Omron CX-Programmer project 新工程 (CX-Programmer 9.73)

# PLC 新PLC1: CS1G-H CPU43

## Global symbols (name address type ; comment)
0.00 BOOL  ; 高压电机启动SB201
0.01 BOOL  ; 高压电机停止SB202
0.02 BOOL  ; 1#高压水泵启动SB203
0.03 BOOL  ; 1#高压水泵停止SB204
0.04 BOOL  ; 1#高压水泵下限SP201
0.05 BOOL  ; 2#高压水泵启动SB205
0.06 BOOL  ; 2#高压水泵停止SB206
0.07 BOOL  ; 2#高压水泵下限SP202
0.08 BOOL  ; 1#润滑油泵启动SB207
0.09 BOOL  ; 1#润滑油泵停止SB208
0.10 BOOL  ; 2#润滑油泵启动SB209
0.11 BOOL  ; 2#润滑油泵停止SB210
0.12 BOOL  ; 前轴承流量下限SP203
0.13 BOOL  ; 后轴承流量下限SP204
0.14 BOOL  ; 前轴承温度上限SP201
0.15 BOOL  ; 后轴承温度上限ST202
100.00 BOOL  ; 断电释放
10.00 BOOL  ; 排料三通阀YV209
10.01 BOOL  ; 防反喷阀进YV203
10.02 BOOL  ; 防反喷阀退YV204
10.03 BOOL  ; 1#断电释放阀YV205
10.04 BOOL  ; 2#断电释放阀YV206
10.05 BOOL  ; 1#蓄压器冲压阀YV207
10.06 BOOL  ; 2#蓄压器冲压阀YV208
10.07 BOOL  ; 搅拌桶下胶电磁阀
10.08 BOOL  ; 1#振动电机M213
10.09 BOOL  ; 原胶搅拌电机M215
10.10 BOOL  ; 输胶泵KA27控制制胶启停
10.12 BOOL  ; 施蜡电机M
10.13 BOOL  ; 施胶泵BPM218
10.14 BOOL  ; 干燥风机停止KA31
10.15 BOOL  ; 干燥风机运行指示
110.00 BOOL  ; Y料位计数启动位
110.05 BOOL  ; 高限料位计数器复
114 CHANNEL  ; 高限料位数据通道
11.00 BOOL  ; 干燥风机电机运行
11.01 BOOL  ; 风机转阀故障灯
11.02 BOOL  ; 干燥风机转阀I
11.03 BOOL  ; 调偏阀2
11.04 BOOL  ; 排污阀
11.05 BOOL  ; 调偏阀1
11.06 BOOL  ; 防火皮带正转
11.07 BOOL  ; 防火皮带反转
11.08 BOOL  ; 干燥风机转阀MII
11.09 BOOL  ; 高压启动指示灯
11.10 BOOL  ; 施胶蜡手动
11.11 BOOL  ; 施胶蜡自动
11.12 BOOL  ; 报警指示
11.13 BOOL  ; 成型料耙运行正常指示灯
11.14 BOOL  ; 高限报警
11.15 BOOL  ; 30%慢、70%中、100%料满常亮
130.00 BOOL  ; 进料螺旋DA启动位
130.01 BOOL  ; 运输螺旋DA启动位
130.03 BOOL  ; 施胶泵DA启动位
134 CHANNEL  ; 施胶泵速度控制通
16.07 BOOL  ; 料耙在运行（来自成型线）
1.00 BOOL  ; 前轴承油压下限SP205
1.01 BOOL  ; 后轴承油压下限SP206
1.02 BOOL  ; 加压油泵启动SB211
1.03 BOOL  ; 加压油泵停止SB212
1.04 BOOL  ; 蓄压器充压泵启动SB213
1.05 BOOL  ; 蓄压器充压泵停止SB214
1.06 BOOL  ; 1#蓄压器充压泵下限SP207
1.07 BOOL  ; 1#蓄压器充压泵上限SP207
1.08 BOOL  ; 2#蓄压器充压泵下限SP208
1.09 BOOL  ; 2#蓄压器充压泵上限SP208
1.10 BOOL  ; 高压注油电机启动SB215
1.11 BOOL  ; 高压注油电机停止SB216
1.12 BOOL  ; 1#油箱液位下限SL201
1.13 BOOL  ; 2#油箱液位下限SL202
1.14 BOOL  ; 压差信号1加压
1.15 BOOL  ; 高压柜故障（来自高压柜）
200 CHANNEL  ; 移位
20.01 BOOL  ; 热磨主电机工作条
20.02 BOOL  ; 放油时间无效T3
20.11 BOOL  ; 蓄压器冲压泵启动位
20.12 BOOL  ; 蓄压器手动冲压
211.00 BOOL  ; 上限
211.01 BOOL  ; 下限
21.00 BOOL  ; 运输螺旋低速极限
21.01 BOOL  ; 运输螺旋高速极限
21.02 BOOL  ; 运输螺旋非正常加
22.00 BOOL  ; 进料螺旋低速极限
22.01 BOOL  ; 进料螺旋高速极限
22.02 BOOL  ; 进料螺旋非正常加
23.00 BOOL  ; 料空值限幅
23.01 BOOL  ; 料满值限幅
23.02 BOOL  ; 最大百分数限制
24.00 BOOL  ; 手动换向开
24.01 BOOL  ; 计量桶已在上限
24.02 BOOL  ; 停
24.03 BOOL  ; 施胶泵低速极限
24.04 BOOL  ; 施胶泵高速极限
24.05 BOOL  ; 施胶泵非正常加减
26.00 BOOL  ; 干燥准备完成
26.01 BOOL  ; 干燥转阀检测脉冲
26.02 BOOL  ; 干燥风机工作位
26.03 BOOL  ; 防火螺旋转阀检测
26.04 BOOL  ; 干燥转阀检测脉冲
26.07 BOOL  ; 停止
2.00 BOOL  ; 拨料电机启动SB217
2.01 BOOL  ; 拨料电机停止SB218
2.02 BOOL  ; 进料螺旋准备完成（来自直流柜）
2.03 BOOL  ; 进料螺旋运行正常（来自直流柜）
2.04 BOOL  ; 升降电机升SB219
2.05 BOOL  ; 升降电机降SB220
2.06 BOOL  ; 料位停止
2.07 BOOL  ; 进料螺旋启动SB222
2.08 BOOL  ; 进料螺旋停止SB223
2.09 BOOL  ; 运输螺旋准备完成（来自直流柜）
2.10 BOOL  ; 运输螺旋运行正常（来自直流柜）
2.11 BOOL  ; 运料螺旋启动
2.12 BOOL  ; 运输螺旋停止SB225
2.13 BOOL  ; 主轴进纽
2.14 BOOL  ; 主轴退钮SA201
2.15 BOOL  ; 排污启动
30 CHANNEL  ; 第一个故障字
30.01 BOOL  ; #1
30.02 BOOL  ; #2
30.03 BOOL  ; #3
30.04 BOOL  ; #4
30.05 BOOL  ; #5
30.06 BOOL  ; #6
30.07 BOOL  ; #7
30.08 BOOL  ; #8
30.09 BOOL  ; #9
30.10 BOOL  ; #10
30.11 BOOL  ; #11
30.12 BOOL  ; #12
30.13 BOOL  ; #13
30.14 BOOL  ; #14
30.15 BOOL  ; #15
31.01 BOOL  ; #16
31.02 BOOL  ; #17
31.03 BOOL  ; #18
31.04 BOOL  ; #19
31.05 BOOL  ; #20
31.06 BOOL  ; #21
31.07 BOOL  ; #22
31.08 BOOL  ; #23
31.09 BOOL  ; #24
35 CHANNEL  ; 1#故障输出字
3.00 BOOL  ; 压差信号2
3.01 BOOL  ; 压差信号3
3.02 BOOL  ; 防反喷阀手动SA202
3.03 BOOL  ; 防反喷阀自动SA202
3.04 BOOL  ; 校验开关SA203
3.05 BOOL  ; 料空整定SB226
3.06 BOOL  ; 料满整定SB227
3.07 BOOL  ; 干燥手/自动
3.08 BOOL  ; 振动电机启动
3.09 BOOL  ; 振动电机停止
3.10 BOOL  ; 原胶搅拌电机启动SB236
3.11 BOOL  ; 搅拌电机停止
3.12 BOOL  ; 进料螺旋加速SB232
3.13 BOOL  ; 进料螺旋减速SB233
3.14 BOOL  ; 运输螺旋加速SB234
3.15 BOOL  ; 运输螺旋减速SB235
4.00 BOOL  ; 排料三通阀
4.01 BOOL  ; 1#流量计SP
4.02 BOOL  ; 成型料耙运行正常
4.03 BOOL  ; 高压风机故障
4.04 BOOL  ; 施蜡加速
4.05 BOOL  ; 施蜡减速
4.06 BOOL  ; 施蜡启动
4.07 BOOL  ; 施蜡停止
4.08 BOOL  ; 1#振动电机启动SB282
4.09 BOOL  ; 1#振动电机停止SB283
4.10 BOOL  ; 2#流量计
4.11 BOOL  ; 施胶手/自动SA211
4.12 BOOL  ; 施胶泵加速SB245
4.13 BOOL  ; 施胶泵减速SB246
4.14 BOOL  ; 施胶泵启动SB247
4.15 BOOL  ; 施胶泵停止SB248
50.00 BOOL  ; 1#巡检通道巡检结束
50.01 BOOL  ; 巡检到1#故障字有故障发生
50.02 BOOL  ; 巡检到2#故障字有故障发生
50.05 BOOL  ; 已确认有故障
50.06 BOOL  ; 运行期间故障保存
50.07 BOOL  ; 报警指示
52.00 BOOL  ; 主机已运行
52.01 BOOL  ; 显示选择
52.02 BOOL  ; 报警复位
52.03 BOOL  ; 主机启动
52.04 BOOL  ; 报警
56.00 BOOL  ; 主机停保持
5.00 BOOL  ; 干燥系统急停SB004
5.01 BOOL  ; 皮带跑偏1
5.02 BOOL  ; 干燥风机启动SB250
5.03 BOOL  ; 干燥风机停止
5.04 BOOL  ; 干燥风机转阀启动SB252I
5.05 BOOL  ; 干燥风机转阀停止SB253
5.08 BOOL  ; 皮带跑偏2
5.09 BOOL  ; 跑偏极限1
5.10 BOOL  ; 防火皮带正转SB258
5.11 BOOL  ; 防火皮带反转SB259
5.12 BOOL  ; 防火皮带停止SB260
5.13 BOOL  ; 风机转阀启动II
5.14 BOOL  ; 风机转阀停止II
5.15 BOOL  ; 跑偏极限2
62.05 BOOL  ; 故障复位信号
66.00 BOOL  ; 防火皮带运行GD
6.00 BOOL  ; 干燥风机风门已关SQ203
6.02 BOOL  ; 高压电机已合闸(来自高压柜）
6.03 BOOL  ; 干燥转阀检测SJ206
6.06 BOOL  ; 干燥转阀II检测GD
6.07 BOOL  ; 料耙运行正常2
6.08 BOOL  ; 高压电机在运行
6.09 BOOL  ; 防火皮带运行检测SJ207
6.11 BOOL  ; 热磨过载信号QF
6.12 BOOL  ; 施胶蜡过载信号QF
6.13 BOOL  ; 压缩空气正常热磨
6.14 BOOL  ; 干燥过载信号QF
6.15 BOOL  ; 报警复位SB281
70.00 BOOL  ; 施胶加速上限
70.01 BOOL  ; 施胶减速下限
75.09 BOOL  ; 主机突停
77.00 BOOL  ; 主轴RUNNING
77.07 BOOL  ; 无胶
78.00 BOOL  ; 干燥风机启动条件
7.00 BOOL  ; 1#滤网
7.01 BOOL  ; 2#滤网
7.02 BOOL  ; 3#滤网
7.03 BOOL  ; 4#滤网
7.04 BOOL  ; 1#输胶启动
7.05 BOOL  ; 1#输胶停止
7.06 BOOL  ; 成型压缩空气正常
7.07 BOOL  ; 搅拌桶放料SB旋钮
7.08 BOOL  ; 搅拌桶下限
7.09 BOOL  ; 搅拌上限
7.12 BOOL  ; 70%料位
7.13 BOOL  ; 成型料仓100%料位
7.14 BOOL  ; 2#输胶启动
7.15 BOOL  ; 2#输胶停止
80.00 BOOL  ; 进料螺旋加速上限
80.01 BOOL  ; 进料螺旋加速下限
80.02 BOOL  ; 运输螺旋加速上限
80.03 BOOL  ; 运输螺旋减速下限
80.15 BOOL  ; 禁止负数
86.00 BOOL  ; 气阀运行位
8.02 BOOL  ; 冷却水流量低
8.03 BOOL  ; 进料螺旋冷却水低
90.00 BOOL  ; 施蜡加速上限
90.01 BOOL  ; 施蜡减速下限
9.00 BOOL  ; 高压主电机启动
9.01 BOOL  ; 主电机停止KA1
9.02 BOOL  ; 1#高压水泵M202
9.03 BOOL  ; 2#高压水泵M203
9.04 BOOL  ; 1#润滑泵M204
9.05 BOOL  ; 2#润滑泵M205
9.06 BOOL  ; 加压油泵M206
9.07 BOOL  ; 蓄压气充压油泵M207
9.08 BOOL  ; 高压注油电机M208
9.09 BOOL  ; 进料螺旋启动KA10
9.10 BOOL  ; 运输螺旋M
9.11 BOOL  ; 拨料电机M209
9.12 BOOL  ; 料位升降电机升M210
9.13 BOOL  ; 料位升降电机降M210
9.14 BOOL  ; 主轴进电磁阀YV202
9.15 BOOL  ; 主轴退电磁阀YV201
C0020 BOOL  ; 转阀检测故障
C0022 BOOL  ; 防火螺旋检测故障
D0 CHANNEL  ; 当前故障显示
D1 CHANNEL  ; 故障信息保存
D100 CHANNEL  ; 工作料位实际值
D102 CHANNEL  ; 工作料位料满值
D104 CHANNEL  ; 工作料位料空值
D106 CHANNEL  ; 工作料位百分比计
D108 CHANNEL  ; 工作料位百分比计
D110 CHANNEL  ; 工作料位百分比计
D1100 CHANNEL  ; F
D1101 CHANNEL  ; 100
D112 CHANNEL  ; 工作料位百分数
D124 CHANNEL  ; 显示器
D200 CHANNEL  ; 料位值存取区
D300 CHANNEL  ; 蓄压压力实时数据�
D70 CHANNEL  ; 1#故障字缓存区
D72 CHANNEL  ; 2#故障字缓存区
D74 CHANNEL  ; 巡检故障信息缓存区
H0 CHANNEL  ; 运输螺旋速度给定
H1 CHANNEL  ; 存储运输螺旋速度
H15 CHANNEL  ; 1#巡检通道
H15.00 BOOL  ; 故障信号寻检
H16 CHANNEL  ; 2#巡检通道
H16.00 BOOL  ; 故障信号寻检
H16.10 BOOL  ; 移位循环结束
H16.11 BOOL  ; 移位循环结束
H4 CHANNEL  ; 进料螺旋速度给定
H9 CHANNEL  ; 存储手动施胶速度
T0000 BOOL  ; 主电机启动完成时间
T0001 BOOL  ; 放油时间确认无效
T0002 BOOL  ; 将胶筒中胶放净
T0003 BOOL  ; 停机放油时间
T0004 BOOL  ; 加减速速率
T0006 BOOL  ; 周期扫描
T0007 BOOL  ; 主机启动完成
T0010 BOOL  ; 料位计数时间
T0011 BOOL  ; 1#计量桶下限位延
T0012 BOOL  ; 延时运行
T0014 BOOL  ; 无故障移位
T0015 BOOL  ; 1#桶上限延时
T0017 BOOL  ; 干燥风机启动延时切断
T0020 BOOL  ; 进料加速延时
T0021 BOOL  ; 加速延时1
T0022 BOOL  ; 1#故障干燥转阀
T0023 BOOL  ; 2#故障干燥转阀II
T0025 BOOL  ; 运输加速延时
T0026 BOOL  ; 加速延时1
T0030 BOOL  ; 延时检测是否仍有
T0031 BOOL  ; 故障显示间隔时间
T0032 BOOL  ; 故障显示间隔时间2
T0033 BOOL  ; 1#高压水低限
T0034 BOOL  ; 2#高压水低限
T0035 BOOL  ; 1#流量计
T0036 BOOL  ; 2#流量计
T0037 BOOL  ; 前轴承流量下限
T0038 BOOL  ; 后轴承流量下限
T0040 BOOL  ; 防火螺旋正转停止运行延时
T0041 BOOL  ; 防火螺旋反转停止运行延时
T0043 BOOL  ; 1#油箱液位
T0045 BOOL  ; 2#油箱液位
T0046 BOOL  ; 5分钟后方可停止运行
T0050 BOOL  ; t
T0051 BOOL  ; t
T0060 BOOL  ; 皮带故障
T0070 BOOL  ; 施蜡加速延时
T0071 BOOL  ; 减速延时1
T0076 BOOL  ; 胶桶下限无胶延时
T0077 BOOL  ; 搅拌桶下限位
T0078 BOOL  ; 胶桶满
T0079 BOOL  ; 胶桶空
T0080 BOOL  ; 施蜡减速延时
T0081 BOOL  ; 减速延时1
T0097 BOOL  ; WHETHER OWN NOW
T0098 BOOL  ; 搅拌桶上限位
T0100 BOOL  ; 延时检测是否仍有
T0250 BOOL  ; 运输加速延时
T0260 BOOL  ; 加速延时1
T0300 BOOL  ; 进料减速延时
T0310 BOOL  ; 减速延时1
T0350 BOOL  ; 运输减速延时
T0360 BOOL  ; 减速延时1
T0400 BOOL  ; 施胶加速延时
T0410 BOOL  ; 加速延时1
T0500 BOOL  ; 施胶减速延时
T0510 BOOL  ; 减速延时1
T1400 BOOL  ; 干燥风机启动延时切断

## Program 新程序1 (cyclic task 0)
; 这个热磨工段自动化控制系统包含热磨主机、运输螺旋、进料螺旋、施胶系统、干燥系统、报警系统和称重系统。通过PLC控制器连接高压电机、水泵、油泵、螺旋输送机、施胶泵、干燥风机、报警装置和称重传感器等系统各个设备。 / 在生产车间中，操作员通过按下高压电机启动按钮启动热磨主机，但前提是1#高压水泵或2#高压水泵、1#润滑油泵和2#润滑油泵已正常运行，同时高压柜无故障信号，确保主机在安全条件下运转。 / 当主电机停止后，1#断电释放阀和2#断电释放阀会自动打开释放压力，保护设备。 / 随后，运输螺旋启动按钮和进料螺旋启动按钮被按下，分别驱动运输螺旋和进料螺旋将木材纤维输送到下一工序。 / 运输螺旋的速度由加速按钮和减速按钮调节，速度设定值始终控制在0到4000之间，避免超速损坏设备。 / 进料螺旋运行时，冷却水流量必须正常，否则进料螺旋不会启动，以防止因冷却不足导致故障。 / 施胶系统通过施胶泵启动按钮激活施胶泵，将胶液均匀涂布在纤维上，其速度由速度设定值控制，且保持在20到4000之间，确保涂布质量。 / 干燥过程由干燥风机启动按钮触发，只有在风门关闭且其他条件满足时，干燥风机才会启动。 / 报警系统通过故障汇总信号监控整个生产线，若检测到异常，报警指示灯会亮起提醒操作员。 / 当故障排除后，操作员需按下报警复位按钮，且故障信号已清零时，报警状态才会复位，确保报警指示灯熄灭，避免误报持续影响生产。 / 称重系统利用当前料位值实时监测物料重量，并通过料位上限信号和料位下限信号确保其在安全范围内，防止物料过载或不足。

### Section 热磨主机

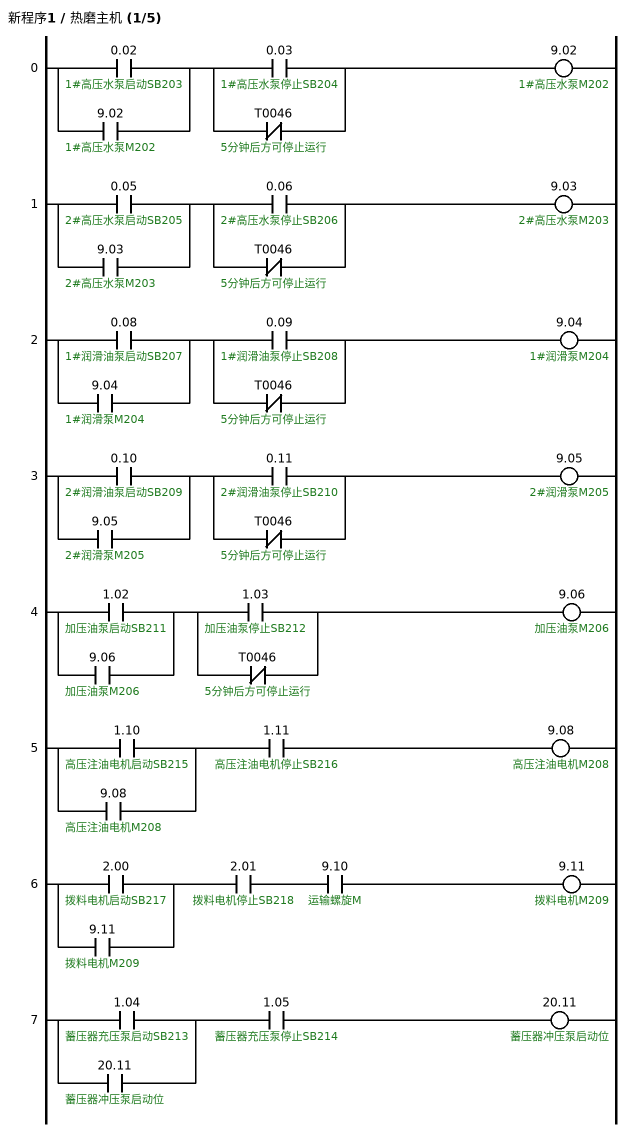
; rung 0
LD 0.02  ; 1#高压水泵启动SB203
OR 9.02  ; 1#高压水泵M202
LD 0.03  ; 1#高压水泵停止SB204
ORNOT T0046  ; 5分钟后方可停止运行
ANDLD
OUT 9.02  ; 1#高压水泵M202
; rung 1
LD 0.05  ; 2#高压水泵启动SB205
OR 9.03  ; 2#高压水泵M203
LD 0.06  ; 2#高压水泵停止SB206
ORNOT T0046  ; 5分钟后方可停止运行
ANDLD
OUT 9.03  ; 2#高压水泵M203
; rung 2
LD 0.08  ; 1#润滑油泵启动SB207
OR 9.04  ; 1#润滑泵M204
LD 0.09  ; 1#润滑油泵停止SB208
ORNOT T0046  ; 5分钟后方可停止运行
ANDLD
OUT 9.04  ; 1#润滑泵M204
; rung 3
LD 0.10  ; 2#润滑油泵启动SB209
OR 9.05  ; 2#润滑泵M205
LD 0.11  ; 2#润滑油泵停止SB210
ORNOT T0046  ; 5分钟后方可停止运行
ANDLD
OUT 9.05  ; 2#润滑泵M205
; rung 4
LD 1.02  ; 加压油泵启动SB211
OR 9.06  ; 加压油泵M206
LD 1.03  ; 加压油泵停止SB212
ORNOT T0046  ; 5分钟后方可停止运行
ANDLD
OUT 9.06  ; 加压油泵M206
; rung 5
LD 1.10  ; 高压注油电机启动SB215
OR 9.08  ; 高压注油电机M208
AND 1.11  ; 高压注油电机停止SB216
OUT 9.08  ; 高压注油电机M208
; rung 6
LD 2.00  ; 拨料电机启动SB217
OR 9.11  ; 拨料电机M209
AND 2.01  ; 拨料电机停止SB218
AND 9.10  ; 运输螺旋M
OUT 9.11  ; 拨料电机M209
; rung 7
LD 1.04  ; 蓄压器充压泵启动SB213
OR 20.11  ; 蓄压器冲压泵启动位
AND 1.05  ; 蓄压器充压泵停止SB214
OUT 20.11  ; 蓄压器冲压泵启动位

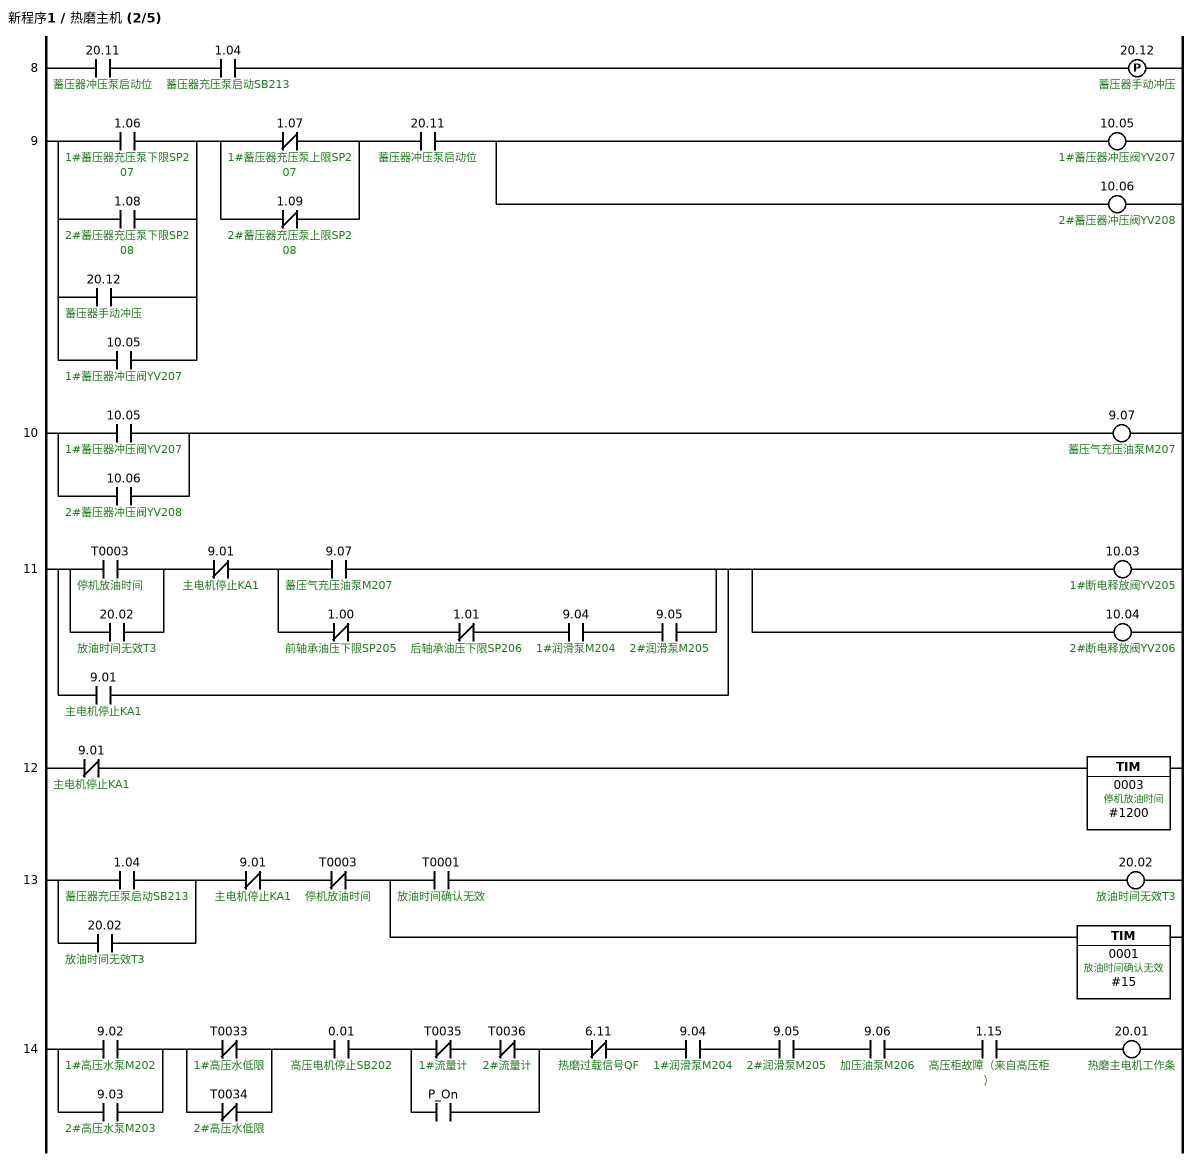
; rung 8
LD 20.11  ; 蓄压器冲压泵启动位
AND 1.04  ; 蓄压器充压泵启动SB213
DIFU(013) 20.12  ; 蓄压器手动冲压
; rung 9
LD 1.06  ; 1#蓄压器充压泵下限SP207
OR 1.08  ; 2#蓄压器充压泵下限SP208
OR 20.12  ; 蓄压器手动冲压
OR 10.05  ; 1#蓄压器冲压阀YV207
LDNOT 1.07  ; 1#蓄压器充压泵上限SP207
ORNOT 1.09  ; 2#蓄压器充压泵上限SP208
ANDLD
AND 20.11  ; 蓄压器冲压泵启动位
OUT 10.05  ; 1#蓄压器冲压阀YV207
OUT 10.06  ; 2#蓄压器冲压阀YV208
; rung 10
LD 10.05  ; 1#蓄压器冲压阀YV207
OR 10.06  ; 2#蓄压器冲压阀YV208
OUT 9.07  ; 蓄压气充压油泵M207
; rung 11
LD T0003  ; 停机放油时间
OR 20.02  ; 放油时间无效T3
ANDNOT 9.01  ; 主电机停止KA1
LD 9.07  ; 蓄压气充压油泵M207
LDNOT 1.00  ; 前轴承油压下限SP205
ANDNOT 1.01  ; 后轴承油压下限SP206
AND 9.04  ; 1#润滑泵M204
AND 9.05  ; 2#润滑泵M205
ORLD
ANDLD
OR 9.01  ; 主电机停止KA1
OUT 10.03  ; 1#断电释放阀YV205
OUT 10.04  ; 2#断电释放阀YV206
; rung 12
LDNOT 9.01  ; 主电机停止KA1
TIM 0003 #1200  ; 停机放油时间
; rung 13
LD 1.04  ; 蓄压器充压泵启动SB213
OR 20.02  ; 放油时间无效T3
ANDNOT 9.01  ; 主电机停止KA1
ANDNOT T0003  ; 停机放油时间
OUT TR0
AND T0001  ; 放油时间确认无效
OUT 20.02  ; 放油时间无效T3
LD TR0
TIM 0001 #15  ; 放油时间确认无效
; rung 14
LD 9.02  ; 1#高压水泵M202
OR 9.03  ; 2#高压水泵M203
LDNOT T0033  ; 1#高压水低限
ORNOT T0034  ; 2#高压水低限
ANDLD
AND 0.01  ; 高压电机停止SB202
LDNOT T0035  ; 1#流量计
ANDNOT T0036  ; 2#流量计
OR P_On
ANDLD
ANDNOT 6.11  ; 热磨过载信号QF
AND 9.04  ; 1#润滑泵M204
AND 9.05  ; 2#润滑泵M205
AND 9.06  ; 加压油泵M206
AND 1.15  ; 高压柜故障（来自高压柜）
OUT 20.01  ; 热磨主电机工作条

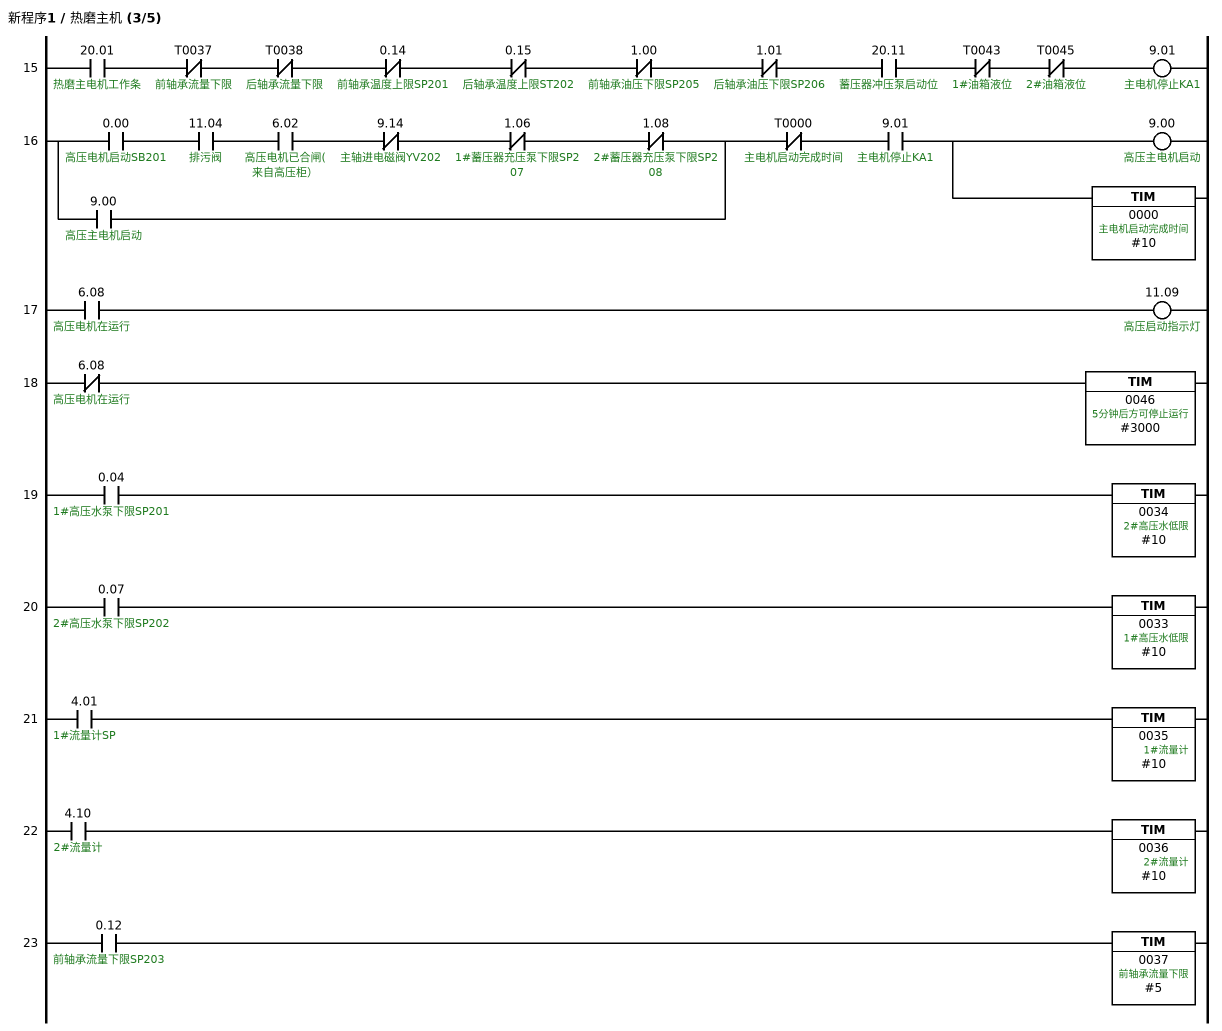
; rung 15
LD 20.01  ; 热磨主电机工作条
ANDNOT T0037  ; 前轴承流量下限
ANDNOT T0038  ; 后轴承流量下限
ANDNOT 0.14  ; 前轴承温度上限SP201
ANDNOT 0.15  ; 后轴承温度上限ST202
ANDNOT 1.00  ; 前轴承油压下限SP205
ANDNOT 1.01  ; 后轴承油压下限SP206
AND 20.11  ; 蓄压器冲压泵启动位
ANDNOT T0043  ; 1#油箱液位
ANDNOT T0045  ; 2#油箱液位
OUT 9.01  ; 主电机停止KA1
; rung 16
LD 0.00  ; 高压电机启动SB201
AND 11.04  ; 排污阀
AND 6.02  ; 高压电机已合闸(来自高压柜）
ANDNOT 9.14  ; 主轴进电磁阀YV202
ANDNOT 1.06  ; 1#蓄压器充压泵下限SP207
ANDNOT 1.08  ; 2#蓄压器充压泵下限SP208
OR 9.00  ; 高压主电机启动
ANDNOT T0000  ; 主电机启动完成时间
AND 9.01  ; 主电机停止KA1
OUT 9.00  ; 高压主电机启动
TIM 0000 #10  ; 主电机启动完成时间
; rung 17
LD 6.08  ; 高压电机在运行
OUT 11.09  ; 高压启动指示灯
; rung 18
LDNOT 6.08  ; 高压电机在运行
TIM 0046 #3000  ; 5分钟后方可停止运行
; rung 19
LD 0.04  ; 1#高压水泵下限SP201
TIM 0034 #10  ; 2#高压水低限
; rung 20
LD 0.07  ; 2#高压水泵下限SP202
TIM 0033 #10  ; 1#高压水低限
; rung 21
LD 4.01  ; 1#流量计SP
TIM 0035 #10  ; 1#流量计
; rung 22
LD 4.10  ; 2#流量计
TIM 0036 #10  ; 2#流量计
; rung 23
LD 0.12  ; 前轴承流量下限SP203
TIM 0037 #5  ; 前轴承流量下限

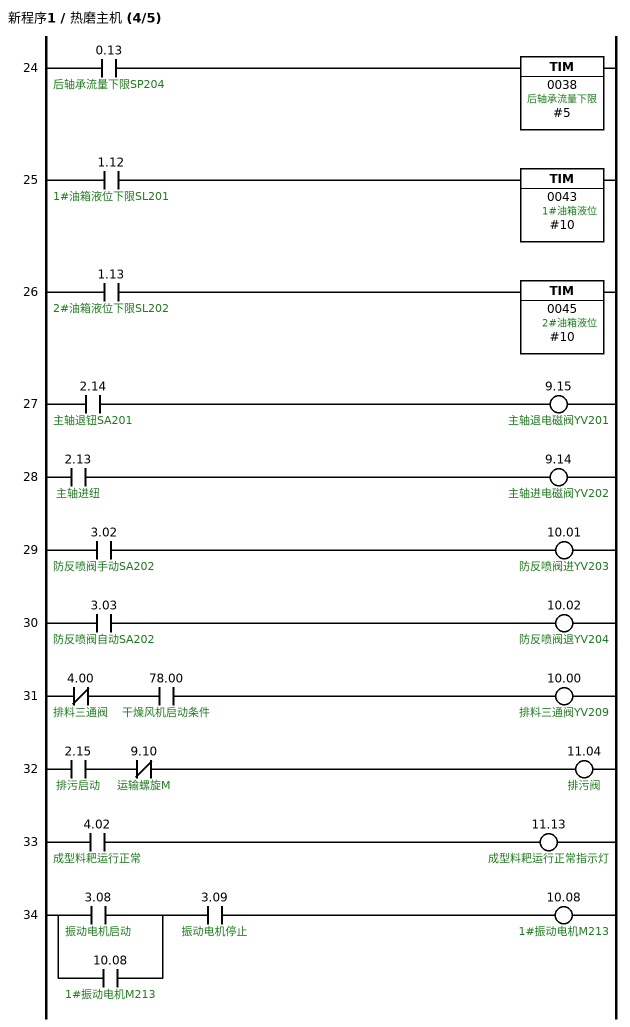
; rung 24
LD 0.13  ; 后轴承流量下限SP204
TIM 0038 #5  ; 后轴承流量下限
; rung 25
LD 1.12  ; 1#油箱液位下限SL201
TIM 0043 #10  ; 1#油箱液位
; rung 26
LD 1.13  ; 2#油箱液位下限SL202
TIM 0045 #10  ; 2#油箱液位
; rung 27
LD 2.14  ; 主轴退钮SA201
OUT 9.15  ; 主轴退电磁阀YV201
; rung 28
LD 2.13  ; 主轴进纽
OUT 9.14  ; 主轴进电磁阀YV202
; rung 29
LD 3.02  ; 防反喷阀手动SA202
OUT 10.01  ; 防反喷阀进YV203
; rung 30
LD 3.03  ; 防反喷阀自动SA202
OUT 10.02  ; 防反喷阀退YV204
; rung 31
LDNOT 4.00  ; 排料三通阀
AND 78.00  ; 干燥风机启动条件
OUT 10.00  ; 排料三通阀YV209
; rung 32
LD 2.15  ; 排污启动
ANDNOT 9.10  ; 运输螺旋M
OUT 11.04  ; 排污阀
; rung 33
LD 4.02  ; 成型料耙运行正常
OUT 11.13  ; 成型料耙运行正常指示灯
; rung 34
LD 3.08  ; 振动电机启动
OR 10.08  ; 1#振动电机M213
AND 3.09  ; 振动电机停止
OUT 10.08  ; 1#振动电机M213

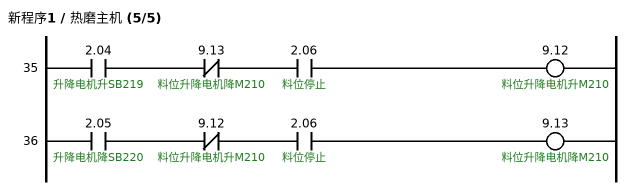
; rung 35
LD 2.04  ; 升降电机升SB219
ANDNOT 9.13  ; 料位升降电机降M210
AND 2.06  ; 料位停止
OUT 9.12  ; 料位升降电机升M210
; rung 36
LD 2.05  ; 升降电机降SB220
ANDNOT 9.12  ; 料位升降电机升M210
AND 2.06  ; 料位停止
OUT 9.13  ; 料位升降电机降M210

### Section 运输螺旋

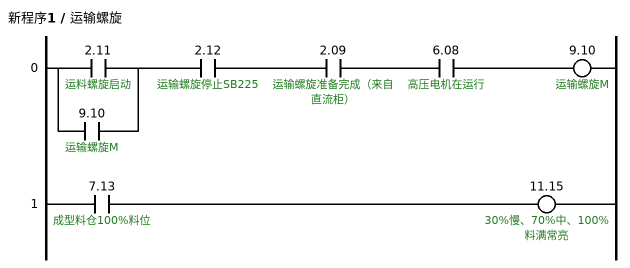
; rung 0
LD 2.11  ; 运料螺旋启动
OR 9.10  ; 运输螺旋M
AND 2.12  ; 运输螺旋停止SB225
AND 2.09  ; 运输螺旋准备完成（来自直流柜）
AND 6.08  ; 高压电机在运行
OUT 9.10  ; 运输螺旋M
; rung 1
LD 7.13  ; 成型料仓100%料位
OUT 11.15  ; 30%慢、70%中、100%料满常亮

### Section 进料螺旋

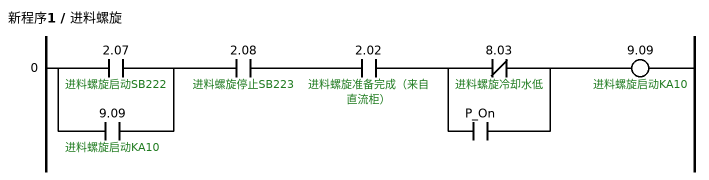
; rung 0
LD 2.07  ; 进料螺旋启动SB222
OR 9.09  ; 进料螺旋启动KA10
AND 2.08  ; 进料螺旋停止SB223
AND 2.02  ; 进料螺旋准备完成（来自直流柜）
LDNOT 8.03  ; 进料螺旋冷却水低
OR P_On
ANDLD
OUT 9.09  ; 进料螺旋启动KA10

### Section 施绞系统

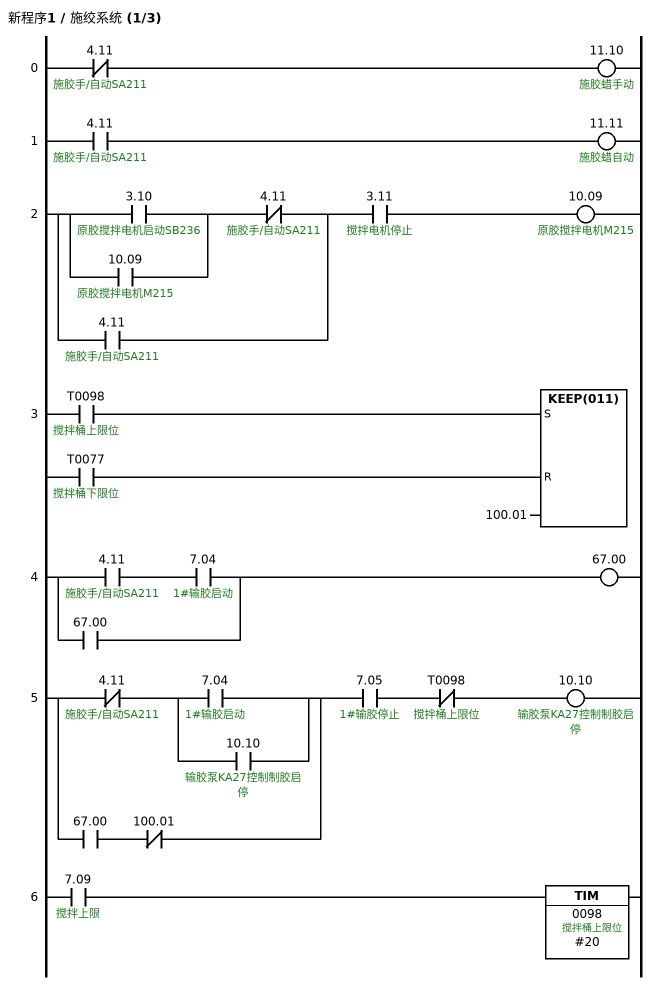
; rung 0
LDNOT 4.11  ; 施胶手/自动SA211
OUT 11.10  ; 施胶蜡手动
; rung 1
LD 4.11  ; 施胶手/自动SA211
OUT 11.11  ; 施胶蜡自动
; rung 2
LD 3.10  ; 原胶搅拌电机启动SB236
OR 10.09  ; 原胶搅拌电机M215
ANDNOT 4.11  ; 施胶手/自动SA211
OR 4.11  ; 施胶手/自动SA211
AND 3.11  ; 搅拌电机停止
OUT 10.09  ; 原胶搅拌电机M215
; rung 3
LD T0098  ; 搅拌桶上限位
LD T0077  ; 搅拌桶下限位
KEEP(011) 100.01
; rung 4
LD 4.11  ; 施胶手/自动SA211
AND 7.04  ; 1#输胶启动
OR 67.00
OUT 67.00
; rung 5
LDNOT 4.11  ; 施胶手/自动SA211
LD 7.04  ; 1#输胶启动
OR 10.10  ; 输胶泵KA27控制制胶启停
ANDLD
LD 67.00
ANDNOT 100.01
ORLD
AND 7.05  ; 1#输胶停止
ANDNOT T0098  ; 搅拌桶上限位
OUT 10.10  ; 输胶泵KA27控制制胶启停
; rung 6
LD 7.09  ; 搅拌上限
TIM 0098 #20  ; 搅拌桶上限位

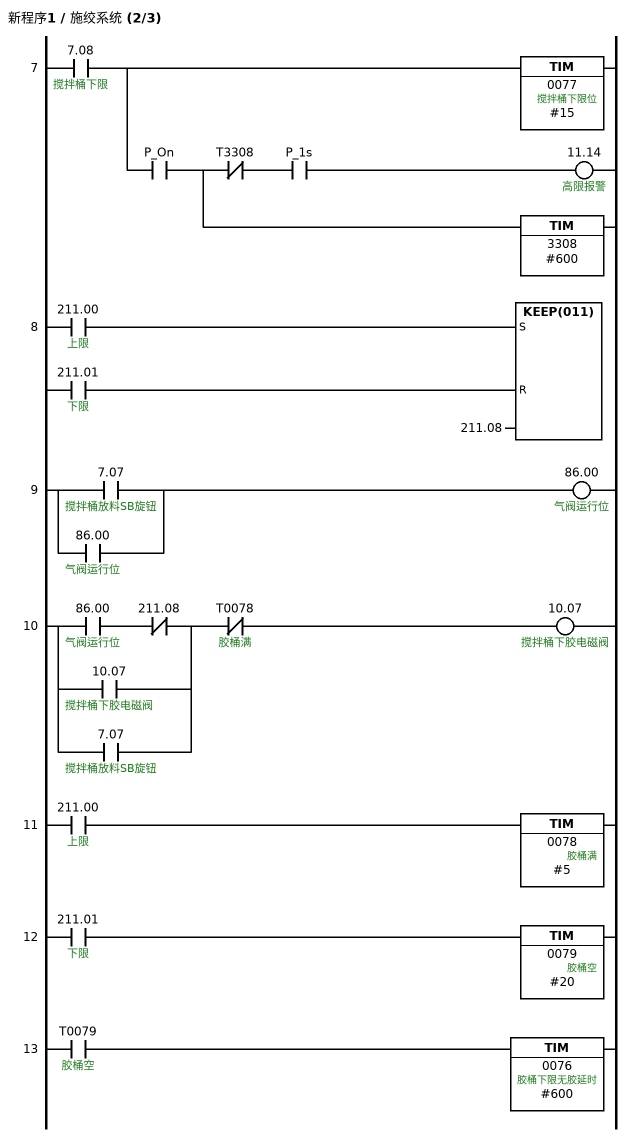
; rung 7
LD 7.08  ; 搅拌桶下限
TIM 0077 #15  ; 搅拌桶下限位
AND P_On
OUT TR0
ANDNOT T3308
AND P_1s
OUT 11.14  ; 高限报警
LD TR0
TIM 3308 #600
; rung 8
LD 211.00  ; 上限
LD 211.01  ; 下限
KEEP(011) 211.08
; rung 9
LD 7.07  ; 搅拌桶放料SB旋钮
OR 86.00  ; 气阀运行位
OUT 86.00  ; 气阀运行位
; rung 10
LD 86.00  ; 气阀运行位
ANDNOT 211.08
OR 10.07  ; 搅拌桶下胶电磁阀
OR 7.07  ; 搅拌桶放料SB旋钮
ANDNOT T0078  ; 胶桶满
OUT 10.07  ; 搅拌桶下胶电磁阀
; rung 11
LD 211.00  ; 上限
TIM 0078 #5  ; 胶桶满
; rung 12
LD 211.01  ; 下限
TIM 0079 #20  ; 胶桶空
; rung 13
LD T0079  ; 胶桶空
TIM 0076 #600  ; 胶桶下限无胶延时

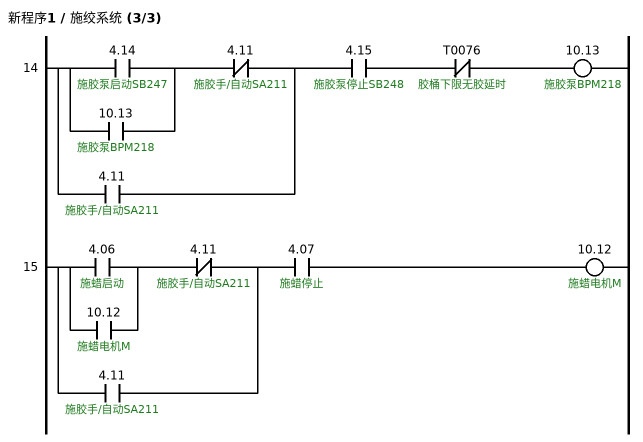
; rung 14
LD 4.14  ; 施胶泵启动SB247
OR 10.13  ; 施胶泵BPM218
ANDNOT 4.11  ; 施胶手/自动SA211
OR 4.11  ; 施胶手/自动SA211
AND 4.15  ; 施胶泵停止SB248
ANDNOT T0076  ; 胶桶下限无胶延时
OUT 10.13  ; 施胶泵BPM218
; rung 15
LD 4.06  ; 施蜡启动
OR 10.12  ; 施蜡电机M
ANDNOT 4.11  ; 施胶手/自动SA211
OR 4.11  ; 施胶手/自动SA211
AND 4.07  ; 施蜡停止
OUT 10.12  ; 施蜡电机M

### Section 报警

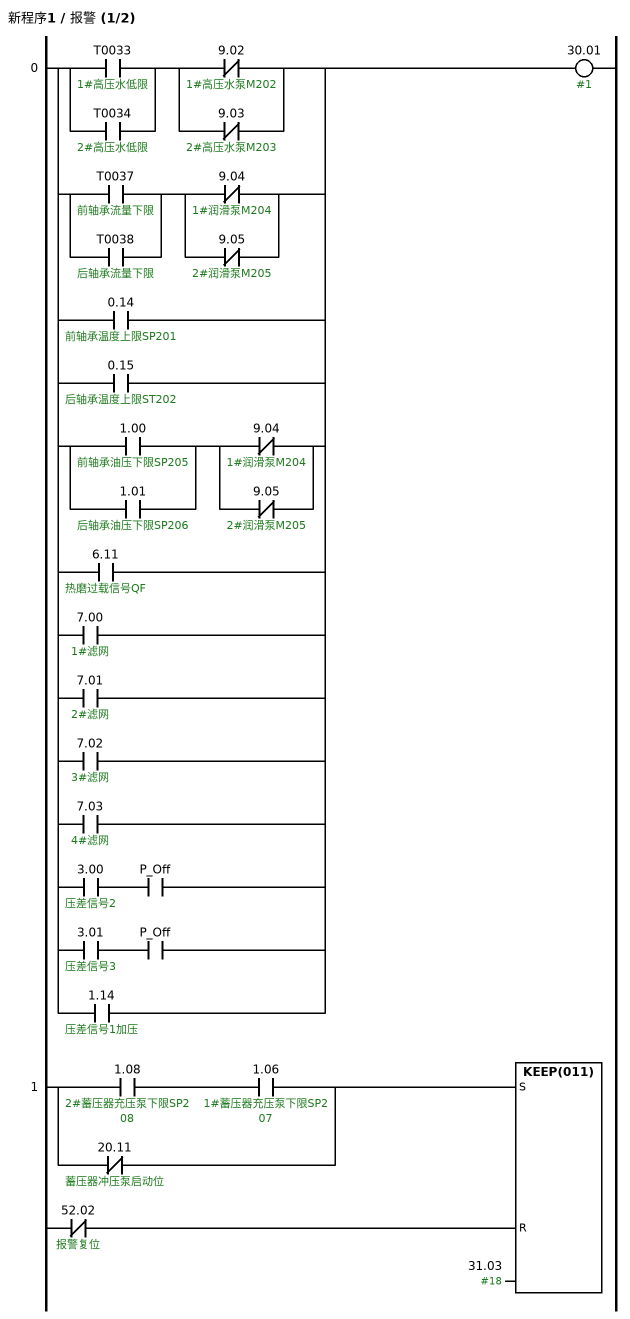
; rung 0
LD T0033  ; 1#高压水低限
OR T0034  ; 2#高压水低限
LDNOT 9.02  ; 1#高压水泵M202
ORNOT 9.03  ; 2#高压水泵M203
ANDLD
LD T0037  ; 前轴承流量下限
OR T0038  ; 后轴承流量下限
LDNOT 9.04  ; 1#润滑泵M204
ORNOT 9.05  ; 2#润滑泵M205
ANDLD
ORLD
OR 0.14  ; 前轴承温度上限SP201
OR 0.15  ; 后轴承温度上限ST202
LD 1.00  ; 前轴承油压下限SP205
OR 1.01  ; 后轴承油压下限SP206
LDNOT 9.04  ; 1#润滑泵M204
ORNOT 9.05  ; 2#润滑泵M205
ANDLD
ORLD
OR 6.11  ; 热磨过载信号QF
OR 7.00  ; 1#滤网
OR 7.01  ; 2#滤网
OR 7.02  ; 3#滤网
OR 7.03  ; 4#滤网
LD 3.00  ; 压差信号2
AND P_Off
ORLD
LD 3.01  ; 压差信号3
AND P_Off
ORLD
OR 1.14  ; 压差信号1加压
OUT 30.01  ; #1
; rung 1
LD 1.08  ; 2#蓄压器充压泵下限SP208
AND 1.06  ; 1#蓄压器充压泵下限SP207
ORNOT 20.11  ; 蓄压器冲压泵启动位
LDNOT 52.02  ; 报警复位
KEEP(011) 31.03  ; #18

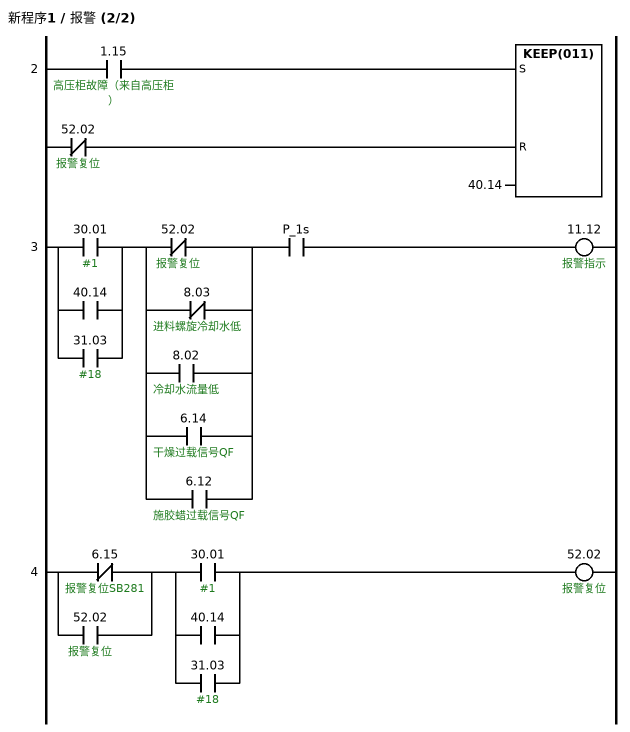
; rung 2
LD 1.15  ; 高压柜故障（来自高压柜）
LDNOT 52.02  ; 报警复位
KEEP(011) 40.14
; rung 3
LD 30.01  ; #1
OR 40.14
OR 31.03  ; #18
LDNOT 52.02  ; 报警复位
ORNOT 8.03  ; 进料螺旋冷却水低
OR 8.02  ; 冷却水流量低
OR 6.14  ; 干燥过载信号QF
OR 6.12  ; 施胶蜡过载信号QF
ANDLD
AND P_1s
OUT 11.12  ; 报警指示
; rung 4
LDNOT 6.15  ; 报警复位SB281
OR 52.02  ; 报警复位
LD 30.01  ; #1
OR 40.14
OR 31.03  ; #18
ANDLD
OUT 52.02  ; 报警复位

### Section 干燥

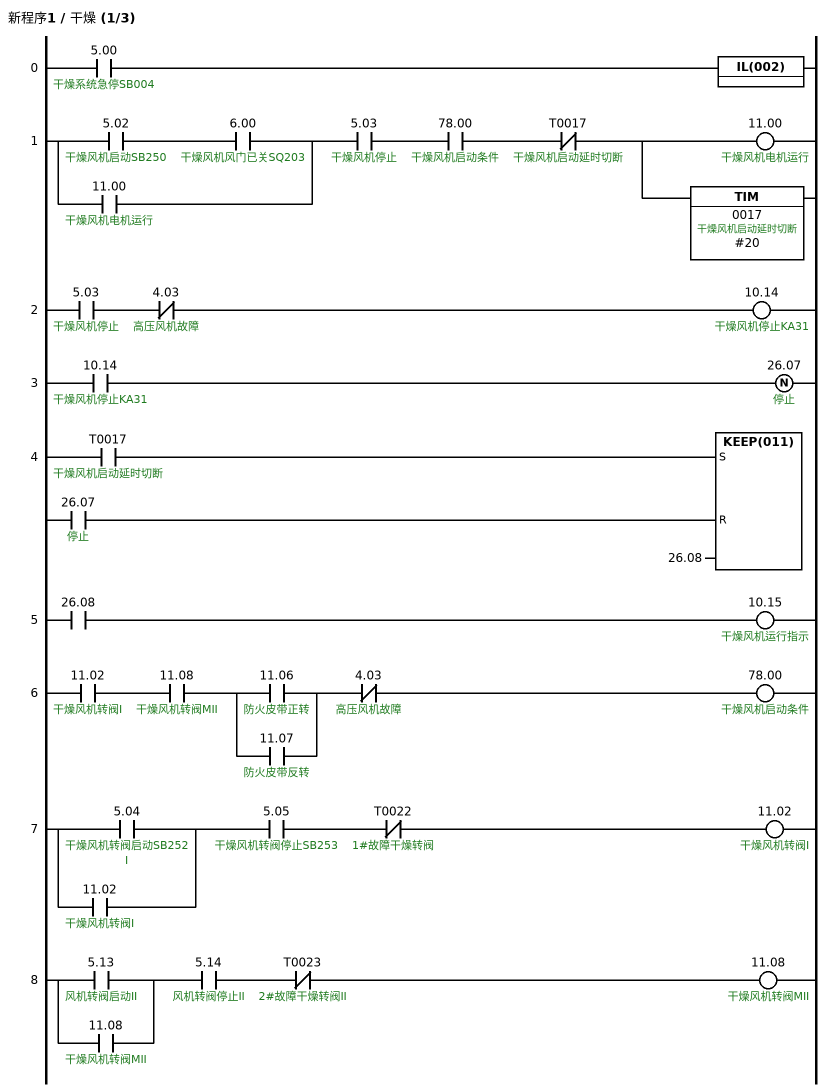
; rung 0
LD 5.00  ; 干燥系统急停SB004
IL(002)
; rung 1
LD 5.02  ; 干燥风机启动SB250
AND 6.00  ; 干燥风机风门已关SQ203
OR 11.00  ; 干燥风机电机运行
AND 5.03  ; 干燥风机停止
AND 78.00  ; 干燥风机启动条件
ANDNOT T0017  ; 干燥风机启动延时切断
OUT 11.00  ; 干燥风机电机运行
TIM 0017 #20  ; 干燥风机启动延时切断
; rung 2
LD 5.03  ; 干燥风机停止
ANDNOT 4.03  ; 高压风机故障
OUT 10.14  ; 干燥风机停止KA31
; rung 3
LD 10.14  ; 干燥风机停止KA31
DIFD(014) 26.07  ; 停止
; rung 4
LD T0017  ; 干燥风机启动延时切断
LD 26.07  ; 停止
KEEP(011) 26.08
; rung 5
LD 26.08
OUT 10.15  ; 干燥风机运行指示
; rung 6
LD 11.02  ; 干燥风机转阀I
AND 11.08  ; 干燥风机转阀MII
LD 11.06  ; 防火皮带正转
OR 11.07  ; 防火皮带反转
ANDLD
ANDNOT 4.03  ; 高压风机故障
OUT 78.00  ; 干燥风机启动条件
; rung 7
LD 5.04  ; 干燥风机转阀启动SB252I
OR 11.02  ; 干燥风机转阀I
AND 5.05  ; 干燥风机转阀停止SB253
ANDNOT T0022  ; 1#故障干燥转阀
OUT 11.02  ; 干燥风机转阀I
; rung 8
LD 5.13  ; 风机转阀启动II
OR 11.08  ; 干燥风机转阀MII
AND 5.14  ; 风机转阀停止II
ANDNOT T0023  ; 2#故障干燥转阀II
OUT 11.08  ; 干燥风机转阀MII

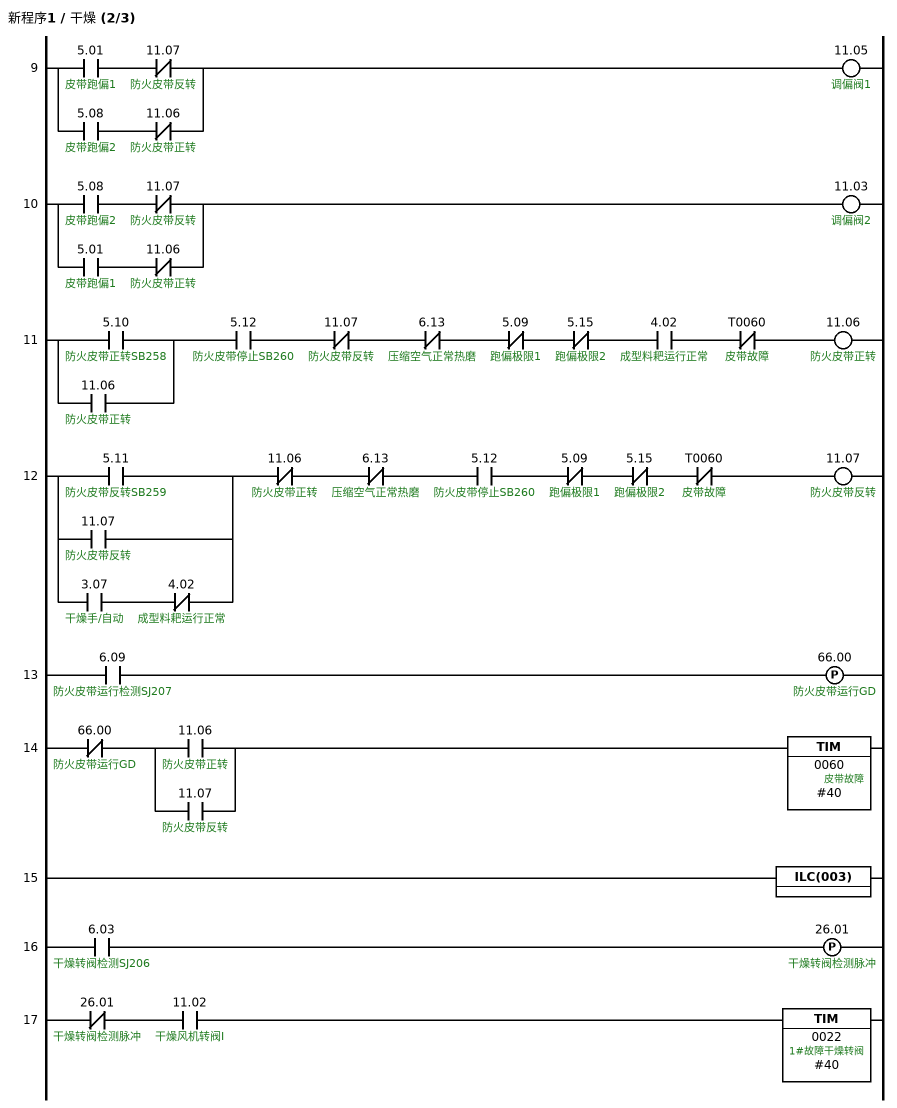
; rung 9
LD 5.01  ; 皮带跑偏1
ANDNOT 11.07  ; 防火皮带反转
LD 5.08  ; 皮带跑偏2
ANDNOT 11.06  ; 防火皮带正转
ORLD
OUT 11.05  ; 调偏阀1
; rung 10
LD 5.08  ; 皮带跑偏2
ANDNOT 11.07  ; 防火皮带反转
LD 5.01  ; 皮带跑偏1
ANDNOT 11.06  ; 防火皮带正转
ORLD
OUT 11.03  ; 调偏阀2
; rung 11
LD 5.10  ; 防火皮带正转SB258
OR 11.06  ; 防火皮带正转
AND 5.12  ; 防火皮带停止SB260
ANDNOT 11.07  ; 防火皮带反转
ANDNOT 6.13  ; 压缩空气正常热磨
ANDNOT 5.09  ; 跑偏极限1
ANDNOT 5.15  ; 跑偏极限2
AND 4.02  ; 成型料耙运行正常
ANDNOT T0060  ; 皮带故障
OUT 11.06  ; 防火皮带正转
; rung 12
LD 5.11  ; 防火皮带反转SB259
OR 11.07  ; 防火皮带反转
LD 3.07  ; 干燥手/自动
ANDNOT 4.02  ; 成型料耙运行正常
ORLD
ANDNOT 11.06  ; 防火皮带正转
ANDNOT 6.13  ; 压缩空气正常热磨
AND 5.12  ; 防火皮带停止SB260
ANDNOT 5.09  ; 跑偏极限1
ANDNOT 5.15  ; 跑偏极限2
ANDNOT T0060  ; 皮带故障
OUT 11.07  ; 防火皮带反转
; rung 13
LD 6.09  ; 防火皮带运行检测SJ207
DIFU(013) 66.00  ; 防火皮带运行GD
; rung 14
LDNOT 66.00  ; 防火皮带运行GD
LD 11.06  ; 防火皮带正转
OR 11.07  ; 防火皮带反转
ANDLD
TIM 0060 #40  ; 皮带故障
; rung 15
ILC(003)
; rung 16
LD 6.03  ; 干燥转阀检测SJ206
DIFU(013) 26.01  ; 干燥转阀检测脉冲
; rung 17
LDNOT 26.01  ; 干燥转阀检测脉冲
AND 11.02  ; 干燥风机转阀I
TIM 0022 #40  ; 1#故障干燥转阀

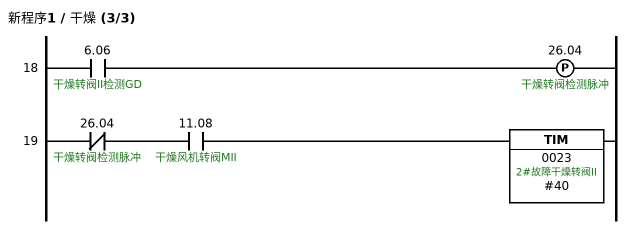
; rung 18
LD 6.06  ; 干燥转阀II检测GD
DIFU(013) 26.04  ; 干燥转阀检测脉冲
; rung 19
LDNOT 26.04  ; 干燥转阀检测脉冲
AND 11.08  ; 干燥风机转阀MII
TIM 0023 #40  ; 2#故障干燥转阀II

### Section 调速

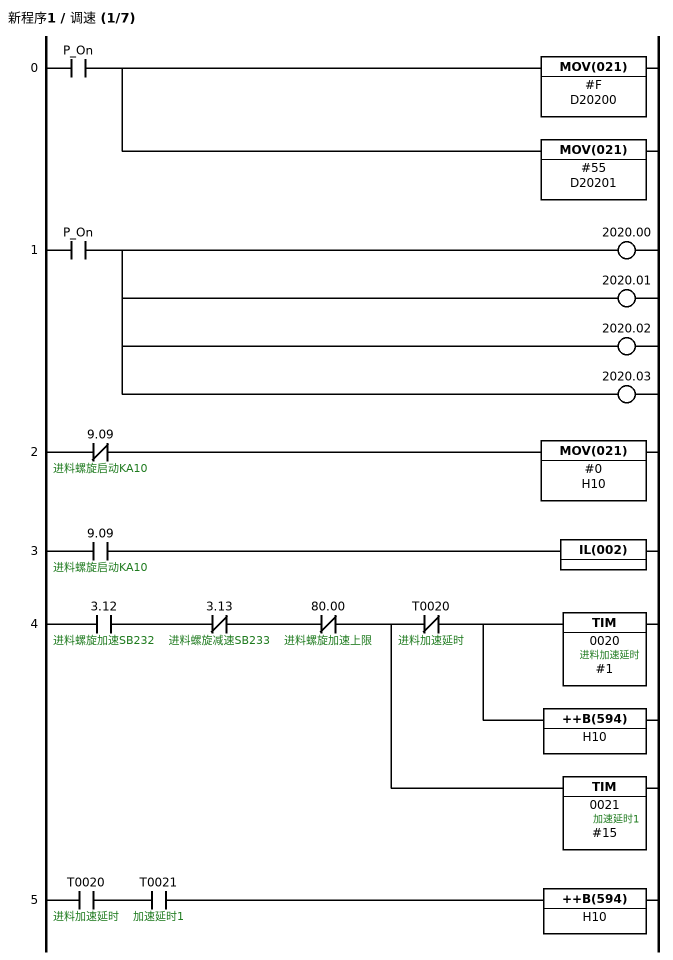
; rung 0
LD P_On
MOV(021) #F D20200
MOV(021) #55 D20201
; rung 1
LD P_On
OUT 2020.00
OUT 2020.01
OUT 2020.02
OUT 2020.03
; rung 2
LDNOT 9.09  ; 进料螺旋启动KA10
MOV(021) #0 H10
; rung 3
LD 9.09  ; 进料螺旋启动KA10
IL(002)
; rung 4
LD 3.12  ; 进料螺旋加速SB232
ANDNOT 3.13  ; 进料螺旋减速SB233
ANDNOT 80.00  ; 进料螺旋加速上限
OUT TR0
ANDNOT T0020  ; 进料加速延时
TIM 0020 #1  ; 进料加速延时
++B(594) H10
LD TR0
TIM 0021 #15  ; 加速延时1
; rung 5
LD T0020  ; 进料加速延时
AND T0021  ; 加速延时1
++B(594) H10

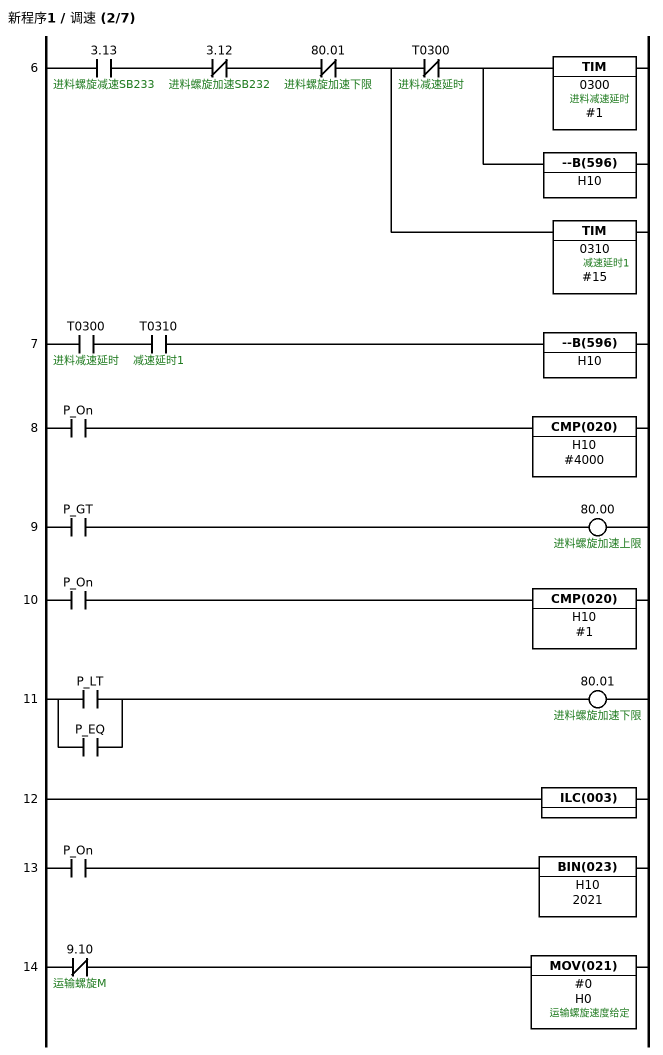
; rung 6
LD 3.13  ; 进料螺旋减速SB233
ANDNOT 3.12  ; 进料螺旋加速SB232
ANDNOT 80.01  ; 进料螺旋加速下限
OUT TR0
ANDNOT T0300  ; 进料减速延时
TIM 0300 #1  ; 进料减速延时
--B(596) H10
LD TR0
TIM 0310 #15  ; 减速延时1
; rung 7
LD T0300  ; 进料减速延时
AND T0310  ; 减速延时1
--B(596) H10
; rung 8
LD P_On
CMP(020) H10 #4000
; rung 9
LD P_GT
OUT 80.00  ; 进料螺旋加速上限
; rung 10
LD P_On
CMP(020) H10 #1
; rung 11
LD P_LT
OR P_EQ
OUT 80.01  ; 进料螺旋加速下限
; rung 12
ILC(003)
; rung 13
LD P_On
BIN(023) H10 2021
; rung 14
LDNOT 9.10  ; 运输螺旋M
MOV(021) #0 H0  ; 运输螺旋速度给定

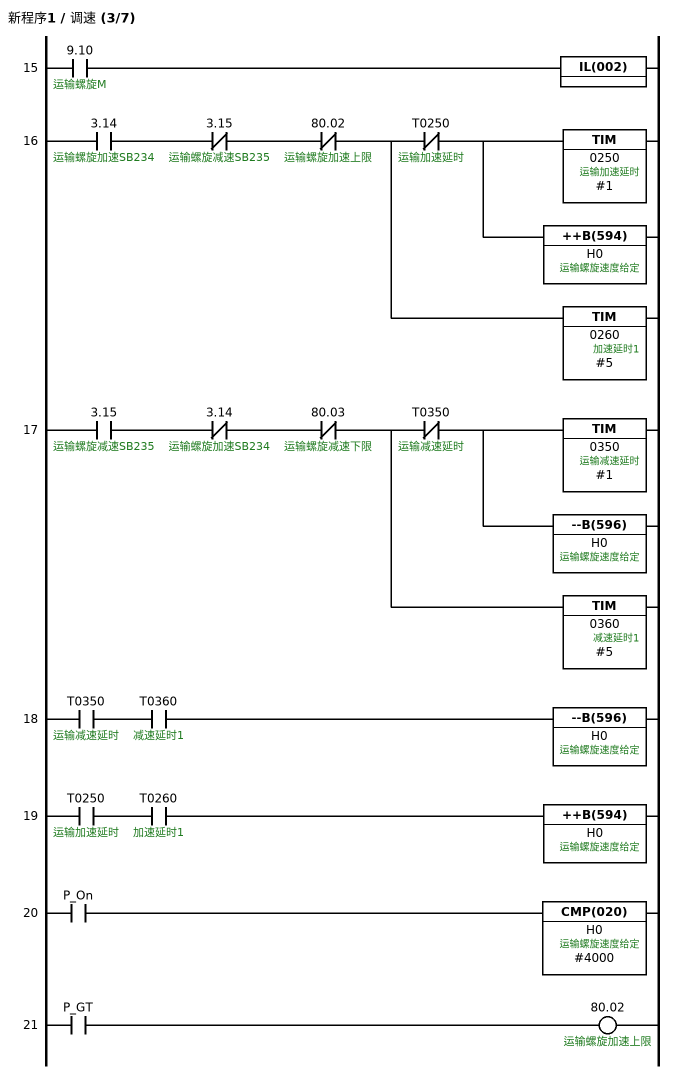
; rung 15
LD 9.10  ; 运输螺旋M
IL(002)
; rung 16
LD 3.14  ; 运输螺旋加速SB234
ANDNOT 3.15  ; 运输螺旋减速SB235
ANDNOT 80.02  ; 运输螺旋加速上限
OUT TR0
ANDNOT T0250  ; 运输加速延时
TIM 0250 #1  ; 运输加速延时
++B(594) H0  ; 运输螺旋速度给定
LD TR0
TIM 0260 #5  ; 加速延时1
; rung 17
LD 3.15  ; 运输螺旋减速SB235
ANDNOT 3.14  ; 运输螺旋加速SB234
ANDNOT 80.03  ; 运输螺旋减速下限
OUT TR0
ANDNOT T0350  ; 运输减速延时
TIM 0350 #1  ; 运输减速延时
--B(596) H0  ; 运输螺旋速度给定
LD TR0
TIM 0360 #5  ; 减速延时1
; rung 18
LD T0350  ; 运输减速延时
AND T0360  ; 减速延时1
--B(596) H0  ; 运输螺旋速度给定
; rung 19
LD T0250  ; 运输加速延时
AND T0260  ; 加速延时1
++B(594) H0  ; 运输螺旋速度给定
; rung 20
LD P_On
CMP(020) H0 #4000  ; 运输螺旋速度给定
; rung 21
LD P_GT
OUT 80.02  ; 运输螺旋加速上限

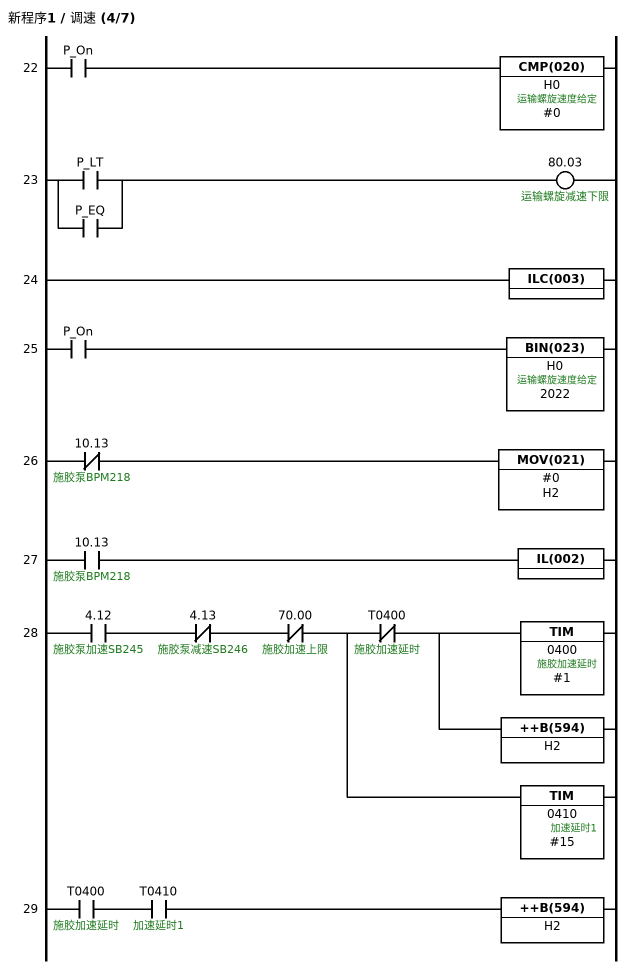
; rung 22
LD P_On
CMP(020) H0 #0  ; 运输螺旋速度给定
; rung 23
LD P_LT
OR P_EQ
OUT 80.03  ; 运输螺旋减速下限
; rung 24
ILC(003)
; rung 25
LD P_On
BIN(023) H0 2022  ; 运输螺旋速度给定
; rung 26
LDNOT 10.13  ; 施胶泵BPM218
MOV(021) #0 H2
; rung 27
LD 10.13  ; 施胶泵BPM218
IL(002)
; rung 28
LD 4.12  ; 施胶泵加速SB245
ANDNOT 4.13  ; 施胶泵减速SB246
ANDNOT 70.00  ; 施胶加速上限
OUT TR0
ANDNOT T0400  ; 施胶加速延时
TIM 0400 #1  ; 施胶加速延时
++B(594) H2
LD TR0
TIM 0410 #15  ; 加速延时1
; rung 29
LD T0400  ; 施胶加速延时
AND T0410  ; 加速延时1
++B(594) H2

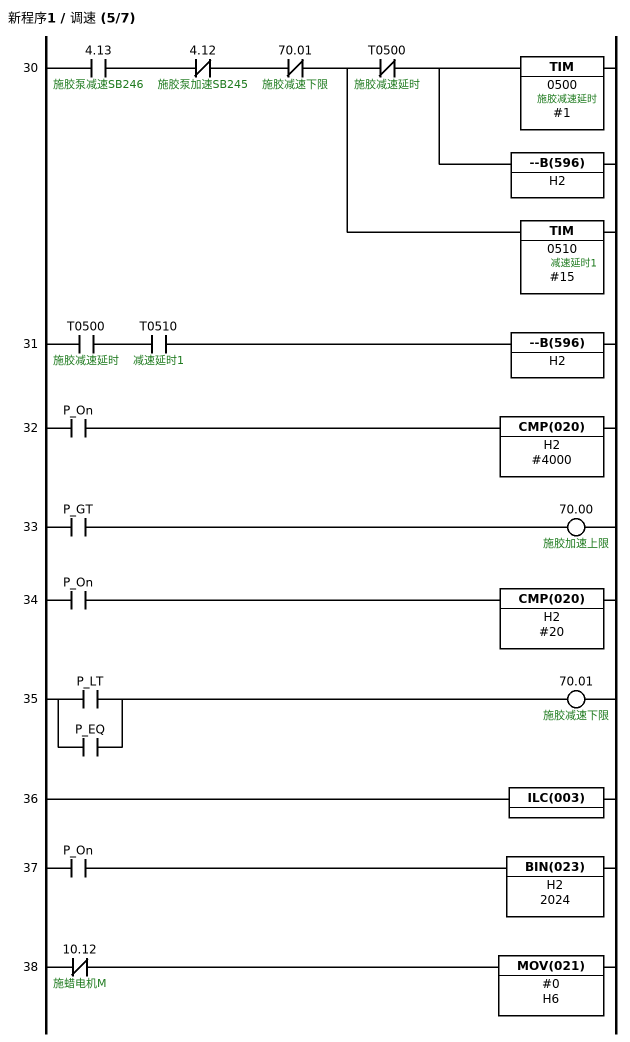
; rung 30
LD 4.13  ; 施胶泵减速SB246
ANDNOT 4.12  ; 施胶泵加速SB245
ANDNOT 70.01  ; 施胶减速下限
OUT TR0
ANDNOT T0500  ; 施胶减速延时
TIM 0500 #1  ; 施胶减速延时
--B(596) H2
LD TR0
TIM 0510 #15  ; 减速延时1
; rung 31
LD T0500  ; 施胶减速延时
AND T0510  ; 减速延时1
--B(596) H2
; rung 32
LD P_On
CMP(020) H2 #4000
; rung 33
LD P_GT
OUT 70.00  ; 施胶加速上限
; rung 34
LD P_On
CMP(020) H2 #20
; rung 35
LD P_LT
OR P_EQ
OUT 70.01  ; 施胶减速下限
; rung 36
ILC(003)
; rung 37
LD P_On
BIN(023) H2 2024
; rung 38
LDNOT 10.12  ; 施蜡电机M
MOV(021) #0 H6

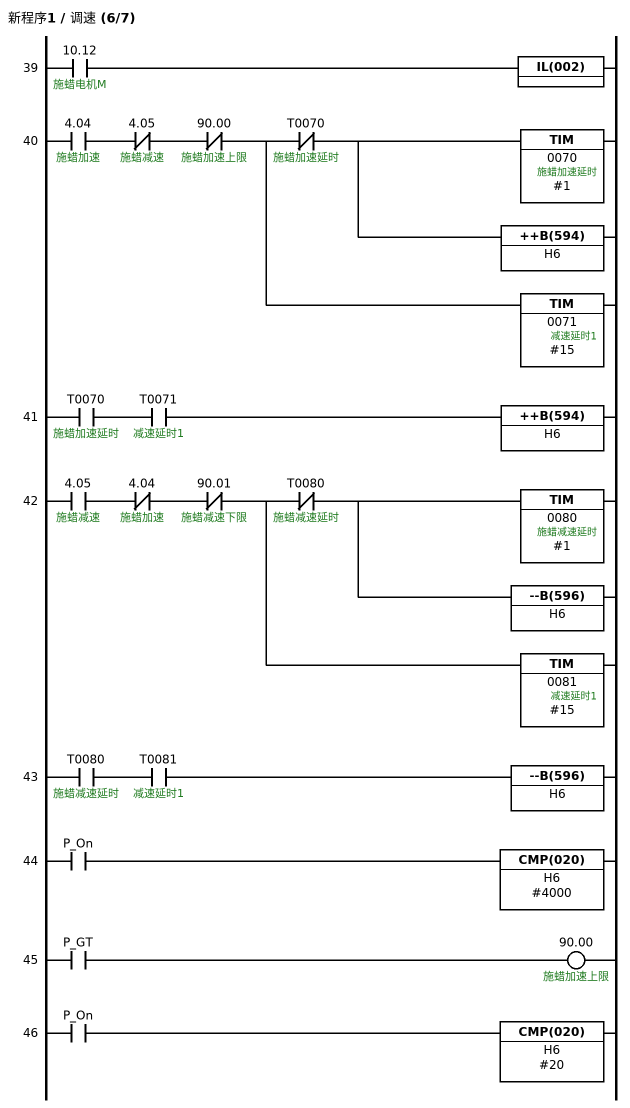
; rung 39
LD 10.12  ; 施蜡电机M
IL(002)
; rung 40
LD 4.04  ; 施蜡加速
ANDNOT 4.05  ; 施蜡减速
ANDNOT 90.00  ; 施蜡加速上限
OUT TR0
ANDNOT T0070  ; 施蜡加速延时
TIM 0070 #1  ; 施蜡加速延时
++B(594) H6
LD TR0
TIM 0071 #15  ; 减速延时1
; rung 41
LD T0070  ; 施蜡加速延时
AND T0071  ; 减速延时1
++B(594) H6
; rung 42
LD 4.05  ; 施蜡减速
ANDNOT 4.04  ; 施蜡加速
ANDNOT 90.01  ; 施蜡减速下限
OUT TR0
ANDNOT T0080  ; 施蜡减速延时
TIM 0080 #1  ; 施蜡减速延时
--B(596) H6
LD TR0
TIM 0081 #15  ; 减速延时1
; rung 43
LD T0080  ; 施蜡减速延时
AND T0081  ; 减速延时1
--B(596) H6
; rung 44
LD P_On
CMP(020) H6 #4000
; rung 45
LD P_GT
OUT 90.00  ; 施蜡加速上限
; rung 46
LD P_On
CMP(020) H6 #20

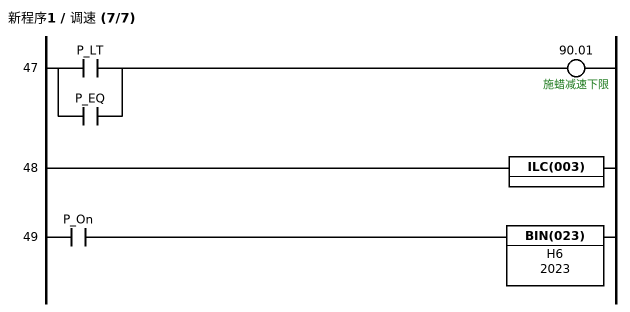
; rung 47
LD P_LT
OR P_EQ
OUT 90.01  ; 施蜡减速下限
; rung 48
ILC(003)
; rung 49
LD P_On
BIN(023) H6 2023

### Section 称重

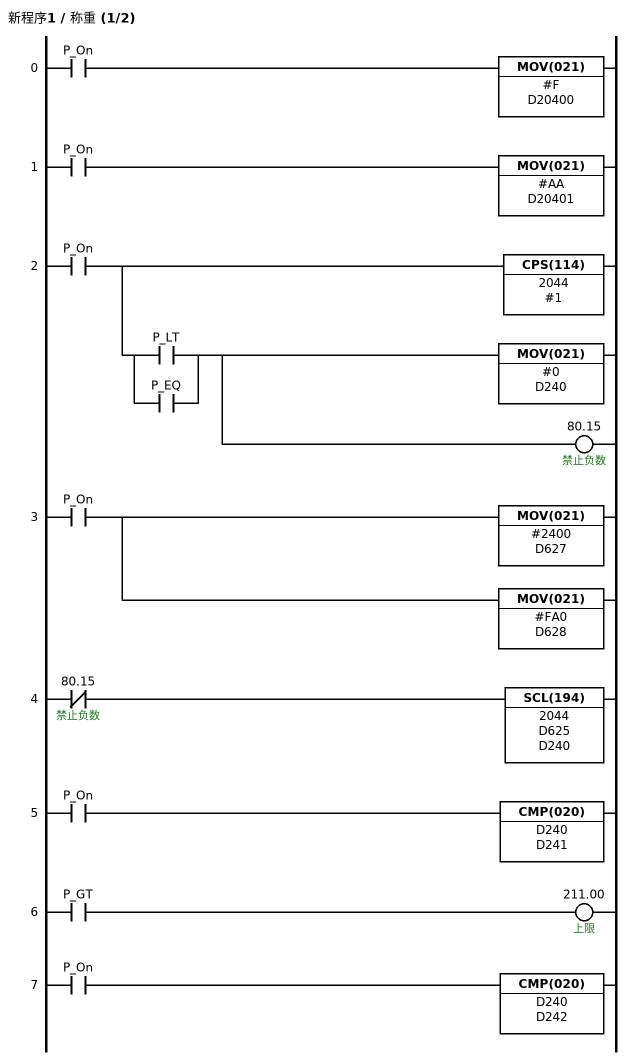
; rung 0
LD P_On
MOV(021) #F D20400
; rung 1
LD P_On
MOV(021) #AA D20401
; rung 2
LD P_On
CPS(114) 2044 #1
LD P_LT
OR P_EQ
ANDLD
MOV(021) #0 D240
OUT 80.15  ; 禁止负数
; rung 3
LD P_On
MOV(021) #2400 D627
MOV(021) #FA0 D628
; rung 4
LDNOT 80.15  ; 禁止负数
SCL(194) 2044 D625 D240
; rung 5
LD P_On
CMP(020) D240 D241
; rung 6
LD P_GT
OUT 211.00  ; 上限
; rung 7
LD P_On
CMP(020) D240 D242

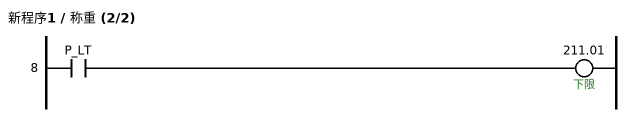
; rung 8
LD P_LT
OUT 211.01  ; 下限

### Section END
; rung 0
END(001)